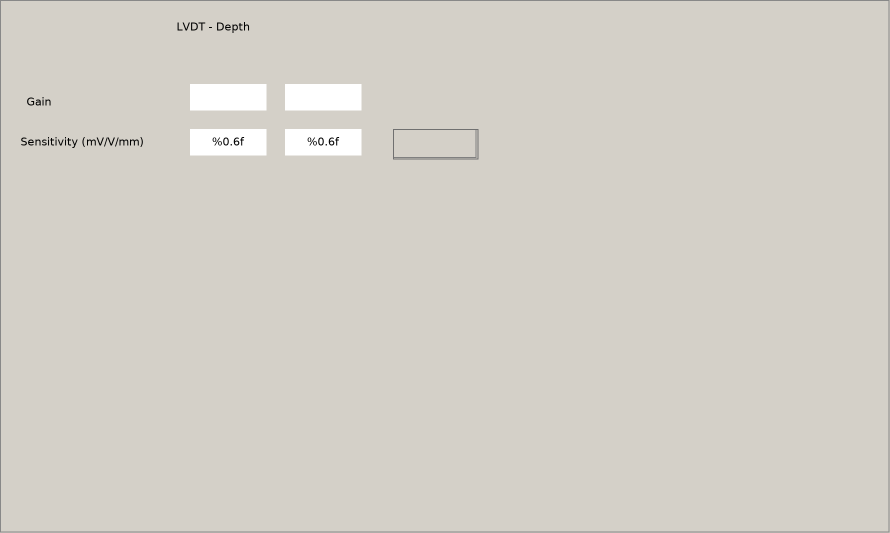
VISUALIZATION V002_CB_Config  // 890x533
    Textfield (284,83 78x28)
    Label (139,12 149x30), "LVDT - Depth"
    Label (11,87 56x30), "Gain"
    Label (15,127 135x30), "Sensitivity (mV/V/mm)"
    Textfield (284,128 78x28), "%0.6f", text variable: Read_Write_CoE.fSensitivity_ToUpload
        OnMouseClick: write Read_Write_CoE.fSensitivity_ToUpload via VisuDialogs.Numpad
    Textfield (189,83 78x28)
    Textfield (189,128 78x28), "%0.6f", text variable: Read_Write_CoE.fSensitivity_Live, input disabled if: TRUE
    Button (393,129 85x30)
        OnMouseDown: toggle Read_Write_CoE.bWriteSensitivity1
        OnMouseUp: toggle Read_Write_CoE.bReadSensitivity1
END_VISUALIZATION

(* stored: Version 1.1.0.1, ProductVersion 3.1.4024.12
   Visu V002_CB_Config: Id {f51c6e8b-4c26-4027-ad0d-fa7f58b10bcc} *)
